Omron Sysmac Studio project Sample_MQTT_Comm_V1_0_0_3 (Sysmac Studio 1.46.0.64007, StandardProject)

# Controller new_Controller_0: NX102-9000 version 1.46

PROGRAM Publisher_Subscriber_LD
VAR
    Trigger : BOOL;
    Operating : BOOL;
    OperatingEnd : BOOL;
    ClientStop : BOOL;
    Execute_ping : BOOL;
    Execue_pub : BOOL;
    Execute_sub : BOOL;
    pubMsg : ARRAY[0..1999] OF BYTE;
    MsgSize : UINT;
    PacketID : UINT;
    MsgType : USINT;
    rcvMsg : ARRAY[0..1999] OF BYTE;
    ElapseTime : UINT;
    info2 : UINT;
    connectionSettings : OmronLib\MQTT_Comm\sConnectionSettings;
    pubFlags : OmronLib\MQTT_Comm\sPubFlags;
    ClientReference : OmronLib\MQTT_Comm\sClientReference;
    MQTTClient_instance : OmronLib\MQTT_Comm\MQTTClient;
    MQTTPing_instance : OmronLib\MQTT_Comm\MQTTPing;
    MQTTPubAryByte_instance : OmronLib\MQTT_Comm\MQTTPubAryByte;
    MQTTSubAryByte_instance : OmronLib\MQTT_Comm\MQTTSubAryByte;
    RS_instance : RS;
END_VAR
VAR_EXTERNAL CONSTANT
    _EIP_EtnOnlineSta : BOOL;
END_VAR
VAR
    _e1 : R_TRIG;
    _e2 : R_TRIG;
    _e3 : R_TRIG;
    _p4 : BOOL;
END_VAR

(* Section Section0: ladder, written here as Structured Text *)

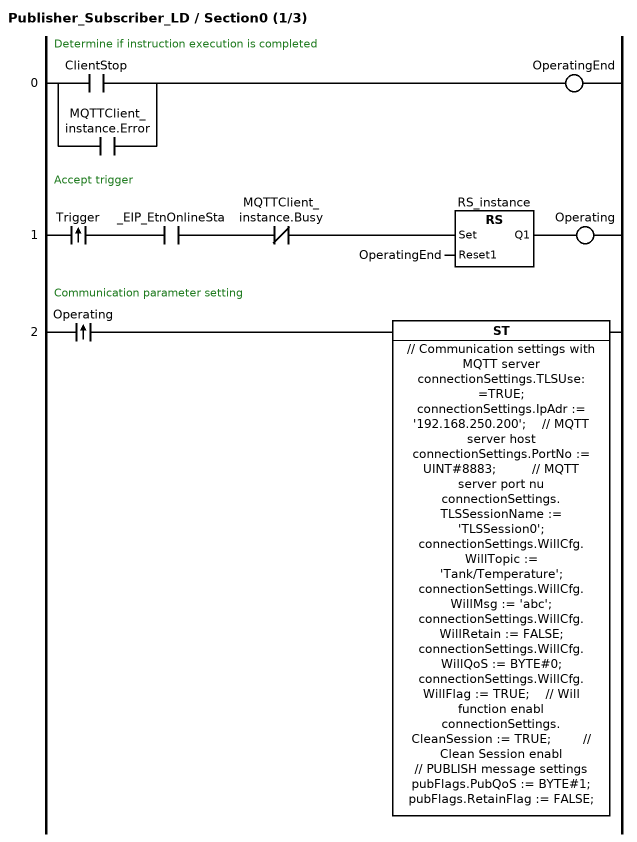
(* Rung 0: Determine if instruction execution is completed *)
OperatingEnd := ClientStop OR MQTTClient_instance.Error;
(* Rung 1: Accept trigger *)
_e1(CLK := Trigger);
RS_instance(Set := _e1.Q AND _EIP_EtnOnlineSta AND NOT MQTTClient_instance.Busy, Reset1 := OperatingEnd);
Operating := RS_instance.Q1;
(* Rung 2: Communication parameter setting *)
_e2(CLK := Operating);
IF _e2.Q THEN
    // Communication settings with MQTT server
    connectionSettings.TLSUse:=TRUE;
    connectionSettings.IpAdr := '192.168.250.200';		// MQTT server host name
    connectionSettings.PortNo := UINT#8883;					// MQTT server port number
    connectionSettings.TLSSessionName := 'TLSSession0';
    connectionSettings.WillCfg.WillTopic := 'Tank/Temperature';
    connectionSettings.WillCfg.WillMsg := 'abc';
    connectionSettings.WillCfg.WillRetain := FALSE;
    connectionSettings.WillCfg.WillQoS := BYTE#0;
    connectionSettings.WillCfg.WillFlag := TRUE;		// Will function enabled
    connectionSettings.CleanSession := TRUE;				// Clean Session enabled
    // PUBLISH message settings
    pubFlags.PubQoS := BYTE#1;
    pubFlags.RetainFlag := FALSE;
END_IF;

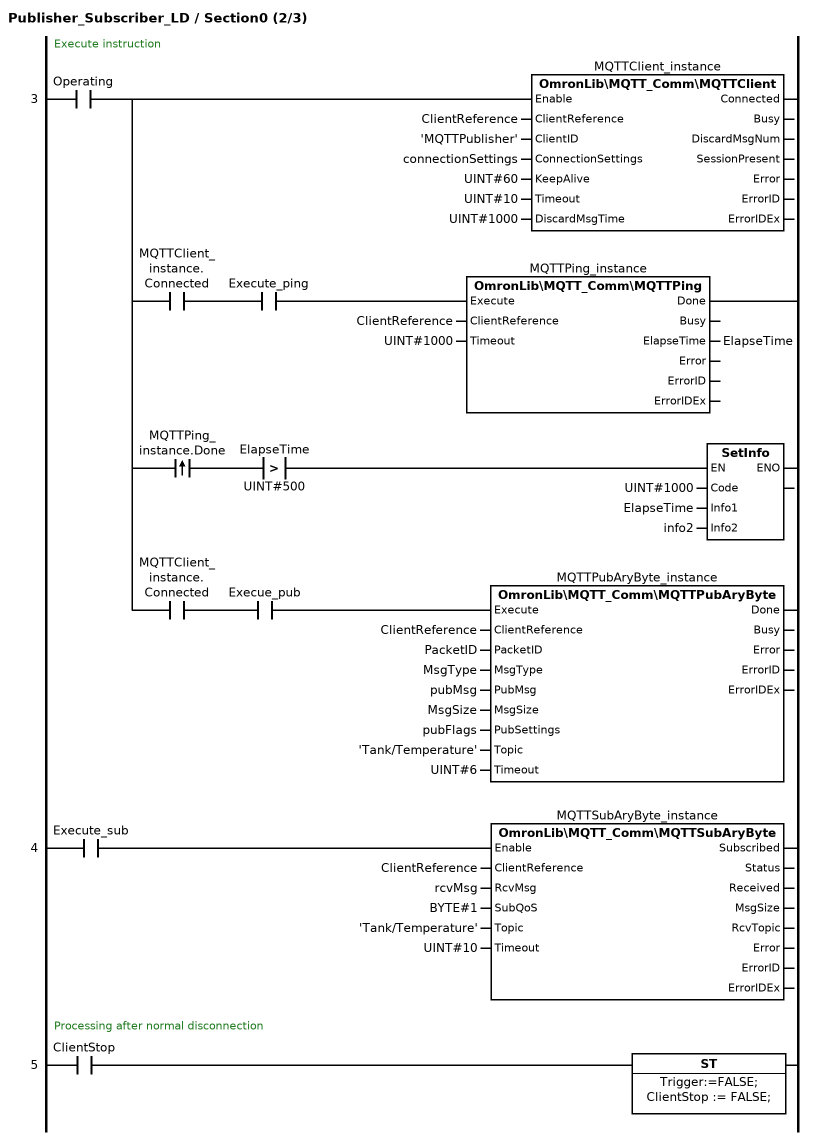
(* Rung 3: Execute instruction *)
MQTTClient_instance(Enable := Operating, ClientReference := ClientReference, ClientID := 'MQTTPublisher', ConnectionSettings := connectionSettings, KeepAlive := UINT#60, Timeout := UINT#10, DiscardMsgTime := UINT#1000);
MQTTPing_instance(Execute := Operating AND MQTTClient_instance.Connected AND Execute_ping, ClientReference := ClientReference, Timeout := UINT#1000, ElapseTime => ElapseTime);
_e3(CLK := MQTTPing_instance.Done);
IF Operating AND _e3.Q AND (ElapseTime > UINT#500) THEN
    SetInfo(Code := UINT#1000, Info1 := ElapseTime, Info2 := info2);
END_IF;
MQTTPubAryByte_instance(Execute := Operating AND MQTTClient_instance.Connected AND Execue_pub, ClientReference := ClientReference, PacketID := PacketID, MsgType := MsgType, PubMsg := pubMsg, MsgSize := MsgSize, PubSettings := pubFlags, Topic := 'Tank/Temperature', Timeout := UINT#6);
(* Rung 4 *)
MQTTSubAryByte_instance(Enable := Execute_sub, ClientReference := ClientReference, RcvMsg := rcvMsg, SubQoS := BYTE#1, Topic := 'Tank/Temperature', Timeout := UINT#10);
(* Rung 5: Processing after normal disconnection *)
_p4 := ClientStop;
IF _p4 THEN
    Trigger:=FALSE;
    ClientStop := FALSE;
END_IF;

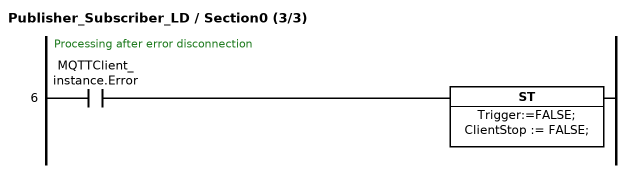
(* Rung 6: Processing after error disconnection *)
IF MQTTClient_instance.Error THEN
    Trigger:=FALSE;
    ClientStop := FALSE;
END_IF;
END_PROGRAM

PROGRAM Publisher_Subscriber_ST
VAR
    Trigger : BOOL;
    DoMQTT : BOOL;
    ClientStop : BOOL;
    Stage : INT;
    Enable_client : BOOL;
    Execute_pub : BOOL;
    Execute_ping : BOOL;
    Enable_subscribe : BOOL;
    pubMsg : ARRAY[0..1999] OF BYTE;
    MsgSize : UINT;
    PacketID : UINT;
    MsgType : USINT;
    connectionSettings : OmronLib\MQTT_Comm\sConnectionSettings := (IpAdr := '', PortNo := 0, TLSUse := False, TLSSessionName := '', UserName := '', Password := '', WillCfg := (WillTopic := '', WillMsg := '', WillRetain := False, WillQoS := 16#0, WillFlag := False), CleanSession := False);
    pubFlags : OmronLib\MQTT_Comm\sPubFlags := (PubQoS := 16#0, RetainFlag := False);
    elapseTime : UINT;
    pingDone : BOOL;
    info2 : UINT;
    rcvMsg : ARRAY[0..1999] OF BYTE;
    ClientReference : OmronLib\MQTT_Comm\sClientReference;
    MQTTClient_instance : OmronLib\MQTT_Comm\MQTTClient;
    MQTTPubAryByte_instance : OmronLib\MQTT_Comm\MQTTPubAryByte;
    MQTTPing_instance : OmronLib\MQTT_Comm\MQTTPing;
    MQTTSubAryByte_instance : OmronLib\MQTT_Comm\MQTTSubAryByte;
    R_TRIG_pingDone : R_TRIG;
END_VAR
VAR_EXTERNAL CONSTANT
    _EIP_EtnOnlineSta : BOOL;
END_VAR
// Preparing for processing
IF  (Trigger = TRUE) AND (DoMQTT = FALSE) AND (_EIP_EtnOnlineSta = TRUE) THEN
	DoMQTT := TRUE;
	Stage := INT#1;
	MQTTClient_instance(Enable := FALSE, ClientReference := ClientReference);			// Initialize instance
	MQTTPing_instance(Execute:=FALSE, ClientReference := ClientReference);		// Initialize instance
	MQTTPubAryByte_instance(																	// Initialize instance
		Execute := FALSE, ClientReference := ClientReference, PacketID:=PacketID, MsgType:=MsgType, PubMsg:=pubMsg);
	// Communication settings with MQTT server
	connectionSettings.TLSUse:=TRUE;
	connectionSettings.IpAdr := '192.168.250.200';		// MQTT server host name
	connectionSettings.PortNo := UINT#8883;					// MQTT server port number
	connectionSettings.TLSSessionName := 'TLSSession0';
	connectionSettings.WillCfg.WillTopic := 'Tank/Temperature';
	connectionSettings.WillCfg.WillMsg := 'abc';
	connectionSettings.WillCfg.WillRetain := TRUE;
	connectionSettings.WillCfg.WillQoS := BYTE#0;
	connectionSettings.WillCfg.WillFlag := FALSE;		// Will function enabled
	connectionSettings.CleanSession := TRUE;				// Clean Session enabled
	// PUBLISH message settings
	pubFlags.PubQoS := BYTE#1;
	pubFlags.RetainFlag := FALSE;
END_IF;

IF (DoMQTT = TRUE) THEN
	CASE Stage OF
	1 :		// Start connection request
		Enable_client := TRUE;
		Stage := INT#2;
		
	2:		// MQTTClient running
		IF ClientStop = TRUE THEN
			Enable_client := FALSE;	// Stop MQTTClient
			Stage := INT#3;
		ELSIF (MQTTClient_instance.Error = TRUE) THEN
			Stage := INT#20;					//  Error occurred
		END_IF;
			
	3:		// Waiting for connection disconnection with MQTT server
		IF MQTTClient_instance.Busy = FALSE THEN
			DoMQTT := FALSE;
			Trigger := FALSE;
			ClientStop := FALSE;
			Stage := INT#10;					//  Normal end
		ELSIF (MQTTClient_instance.Error = TRUE) THEN
			Stage := INT#20;					//  Error occurred
		END_IF;
		
	20:	//  Error End
		Enable_client := FALSE;
		// Wait for all FB to stop running
		IF MQTTClient_instance.Busy = FALSE THEN
			DoMQTT := FALSE;
			Trigger := FALSE;
			ClientStop := FALSE;
		END_IF;
			
	END_CASE;

END_IF;

MQTTClient_instance(
	Enable							:=	Enable_client,
	ClientReference			:= ClientReference,
	ClientID						:= 'MQTTPublisher',
	ConnectionSettings 	:= connectionSettings,
	KeepAlive						:=	UINT#60,
	Timeout						:= UINT#10,
	DiscardMsgTime			:= UINT#1000);

MQTTPing_instance(
	Execute				:= MQTTClient_instance.Connected AND Execute_ping,
	ClientReference   := ClientReference,
	Timeout				:= UINT#1000,
	ElapseTime			=> elapseTime);

R_TRIG_pingDone(MQTTPubAryByte_instance.Done, pingDone);
IF MQTTClient_instance.Connected AND pingDone AND elapseTime > UINT#500
	THEN
		SetInfo(UINT#1000, elapseTime, info2);
END_IF;

MQTTPubAryByte_instance(
	Execute				:= MQTTClient_instance.Connected AND Execute_pub,
	ClientReference   := ClientReference,
	PacketID				:= PacketID,
	MsgType				:= MsgType,
	PubMsg				:= pubMsg,
	MsgSize				:= MsgSize,
	PubSettings			:= pubFlags,
	Topic					:= 'Tank/Temperature',
	Timeout				:= UINT#6);

MQTTSubAryByte_instance(
	Enable					:= Enable_subscribe,
	ClientReference	:= ClientReference,
	rcvMsg					:= rcvMsg,
	SubQoS				:= BYTE#1,
	Topic					:= 'Tank/Temperature',
	Timeout				:= UINT#10);
END_PROGRAM